(* PLC project CoDeSys External Library Template, WAGO e!COCKPIT e!COCKPIT, author 3S - Smart Software Solutions GmbH *)
(* stored: creationDateTime 2019-10-29T12:22:40.5660807, version 3.5.5.30, modificationDateTime 2019-10-24T14:40:07.960949, organization 3S - Smart Software Solutions GmbH *)
(* Library project template with all possible element types, docu and a sample project structure *)

TYPE typKomunikat : STRUCT
  sZnacznik : STRING;
  sTypKomunikatu : STRING;
  sMnemonikWlasciciela : STRING;
  sMnemonikWlascicielaExt : STRING;
  sMACAdres : STRING;
  sIDZrodla : STRING;
  sIDZrodlaLokalizacja : STRING;
  sIDZrodlaUrzadzenie : STRING;
  sIDPrzeznaczenia : STRING;
  sIDPrzeznaczeniaLokalizacja : STRING;
  sIDPrzeznaczeniaUrzadzenie : STRING;
  sDlugoscPolaDanych : STRING;
  sMarkerCzasowy : STRING;
  sRezerwa : STRING;
  sDane : alSTRINGKomunikat;
END_STRUCT;
END_TYPE
